PROGRAM Axis_13_Function_Blocks
VAR
END_VAR

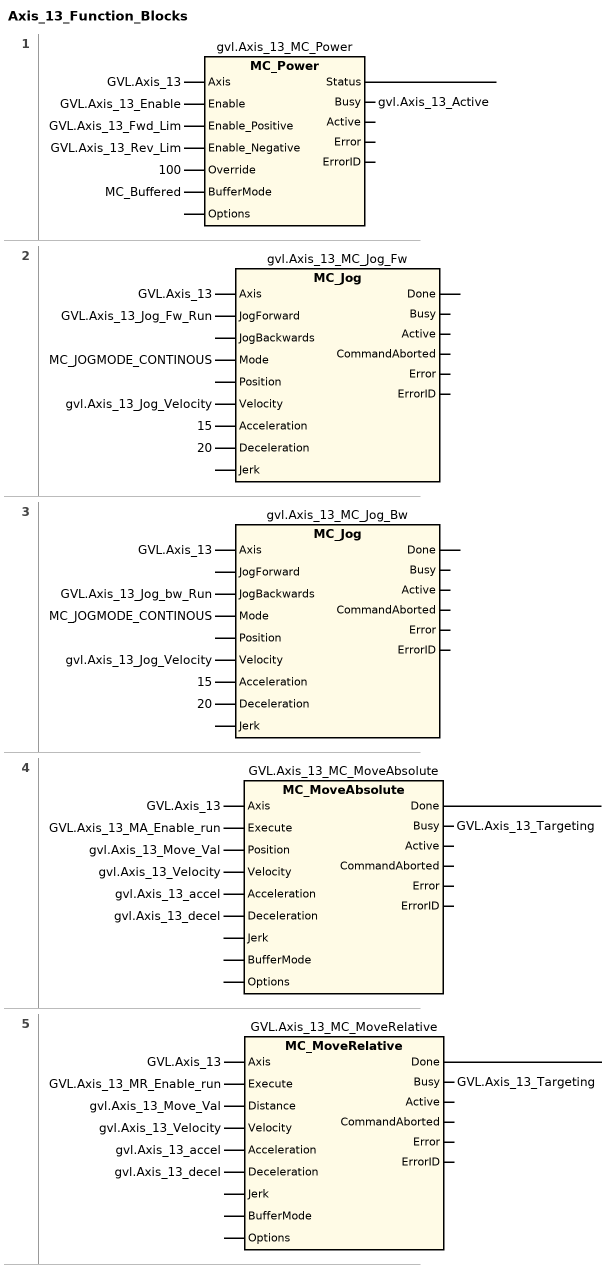
// NETWORK 1
gvl.Axis_13_MC_Power(
    Axis := GVL.Axis_13,
    Enable := GVL.Axis_13_Enable,
    Enable_Positive := GVL.Axis_13_Fwd_Lim,
    Enable_Negative := GVL.Axis_13_Rev_Lim,
    Override := 100,
    BufferMode := MC_Buffered,
    Busy => gvl.Axis_13_Active); // MC_Power

// NETWORK 2
gvl.Axis_13_MC_Jog_Fw(
    Axis := GVL.Axis_13,
    JogForward := GVL.Axis_13_Jog_Fw_Run,
    Mode := MC_JOGMODE_CONTINOUS,
    Velocity := gvl.Axis_13_Jog_Velocity,
    Acceleration := 15,
    Deceleration := 20); // MC_Jog

// NETWORK 3
gvl.Axis_13_MC_Jog_Bw(
    Axis := GVL.Axis_13,
    JogBackwards := GVL.Axis_13_Jog_bw_Run,
    Mode := MC_JOGMODE_CONTINOUS,
    Velocity := gvl.Axis_13_Jog_Velocity,
    Acceleration := 15,
    Deceleration := 20); // MC_Jog

// NETWORK 4
GVL.Axis_13_MC_MoveAbsolute(
    Axis := GVL.Axis_13,
    Execute := GVL.Axis_13_MA_Enable_run,
    Position := gvl.Axis_13_Move_Val,
    Velocity := gvl.Axis_13_Velocity,
    Acceleration := gvl.Axis_13_accel,
    Deceleration := gvl.Axis_13_decel,
    Busy => GVL.Axis_13_Targeting); // MC_MoveAbsolute

// NETWORK 5
GVL.Axis_13_MC_MoveRelative(
    Axis := GVL.Axis_13,
    Execute := GVL.Axis_13_MR_Enable_run,
    Distance := gvl.Axis_13_Move_Val,
    Velocity := gvl.Axis_13_Velocity,
    Acceleration := gvl.Axis_13_accel,
    Deceleration := gvl.Axis_13_decel,
    Busy => GVL.Axis_13_Targeting); // MC_MoveRelative

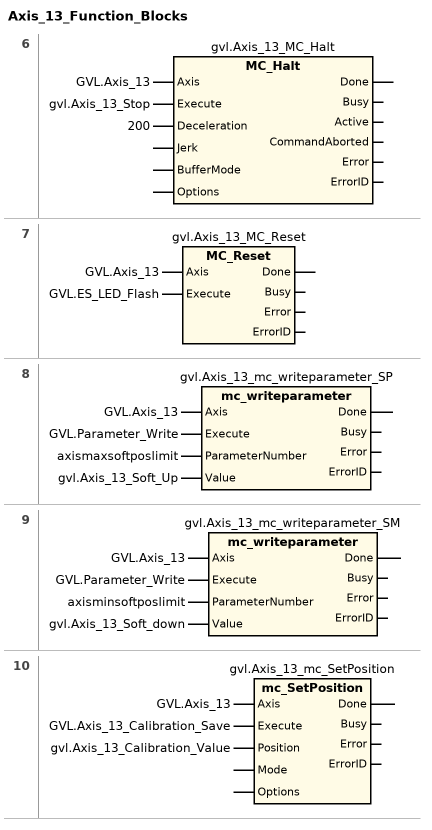
// NETWORK 6
gvl.Axis_13_MC_Halt(Axis := GVL.Axis_13, Execute := gvl.Axis_13_Stop, Deceleration := 200); // MC_Halt

// NETWORK 7
gvl.Axis_13_MC_Reset(Axis := GVL.Axis_13, Execute := GVL.ES_LED_Flash); // MC_Reset

// NETWORK 8
gvl.Axis_13_mc_writeparameter_SP(
    Axis := GVL.Axis_13,
    Execute := GVL.Parameter_Write,
    ParameterNumber := axismaxsoftposlimit,
    Value := gvl.Axis_13_Soft_Up); // mc_writeparameter

// NETWORK 9
gvl.Axis_13_mc_writeparameter_SM(
    Axis := GVL.Axis_13,
    Execute := GVL.Parameter_Write,
    ParameterNumber := axisminsoftposlimit,
    Value := gvl.Axis_13_Soft_down); // mc_writeparameter

// NETWORK 10
gvl.Axis_13_mc_SetPosition(
    Axis := GVL.Axis_13,
    Execute := GVL.Axis_13_Calibration_Save,
    Position := gvl.Axis_13_Calibration_Value); // mc_SetPosition

END_PROGRAM

(* stored: Version 1.1.0.1, ProductVersion 3.1.4022.12
   POU Axis_13_Function_Blocks: Id {2b1eb5fe-9083-40a6-a339-2fc9eba06ed1}, SpecialFunc None *)
